// TIA Portal V18 export
FUNCTION "Re-filling Sequence" : Void   // FC14, LAD
{ S7_Optimized_Access := 'TRUE' }
VERSION : 0.1
// stored: AutoNumber true, IsIECCheckEnabled false, SetENOAutomatically false, UDAEnableTagReadback false
   VAR_TEMP   // added for the SCL form of the ladder/FBD networks
      _w1 : Bool;
      _w2 : Bool;
      _w3 : Bool;
   END_VAR
BEGIN

REGION Network 1
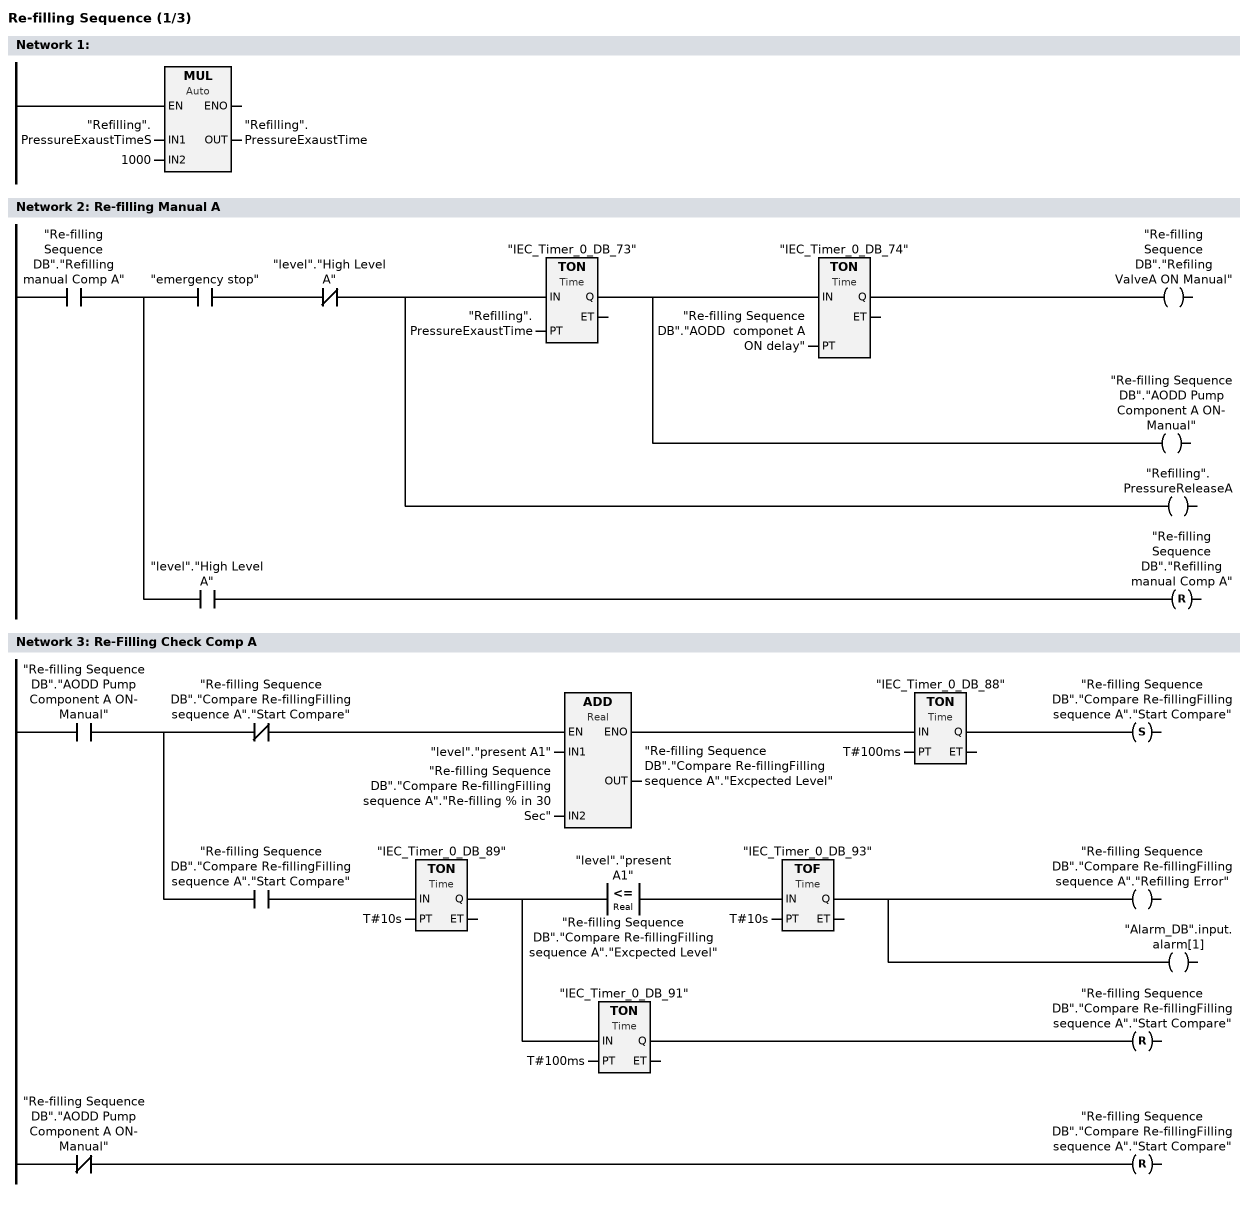
   RUNG wire#powerrail
      Mul(in1 := "Refilling".PressureExaustTimeS, in2 := 1000, out => "Refilling".PressureExaustTime)
   END_RUNG
   // the same network as SCL:
   "Refilling".PressureExaustTime := "Refilling".PressureExaustTimeS * 1000;
END_REGION

REGION Network 2: Re-filling Manual A
   RUNG wire#powerrail
      Contact( "Re-filling Sequence DB"."Refilling manual Comp A" )
      wire#w1
      Contact( "emergency stop" )
      I_Contact( "level"."High Level A" )
      wire#w2
      { S7_Templates := "time_type := Time" } "IEC_Timer_0_DB_73".TON(pt := "Refilling".PressureExaustTime, et =>)
      wire#w3
      { S7_Templates := "time_type := Time" } "IEC_Timer_0_DB_74".TON(pt := "Re-filling Sequence DB"."AODD  componet A  ON delay", et =>)
      Coil( "Re-filling Sequence DB"."Refiling ValveA ON Manual" )
   END_RUNG
   RUNG wire#w3
      Coil( "Re-filling Sequence DB"."AODD Pump Component A ON- Manual" )
   END_RUNG
   RUNG wire#w2
      Coil( "Refilling".PressureReleaseA )
   END_RUNG
   RUNG wire#w1
      Contact( "level"."High Level A" )
      R_Coil( "Re-filling Sequence DB"."Refilling manual Comp A" )
   END_RUNG
   // the same network as SCL:
   #_w1 := "Re-filling Sequence DB"."Refilling manual Comp A" AND "emergency stop" AND NOT "level"."High Level A";
   "IEC_Timer_0_DB_73".TON(IN := #_w1, PT := "Refilling".PressureExaustTime);
   "IEC_Timer_0_DB_74".TON(IN := "IEC_Timer_0_DB_73".Q,
                           PT := "Re-filling Sequence DB"."AODD  componet A  ON delay");
   "Re-filling Sequence DB"."Refiling ValveA ON Manual" := "IEC_Timer_0_DB_74".Q;
   "Re-filling Sequence DB"."AODD Pump Component A ON- Manual" := "IEC_Timer_0_DB_73".Q;
   "Refilling".PressureReleaseA := #_w1;
   IF "Re-filling Sequence DB"."Refilling manual Comp A" AND "level"."High Level A" THEN
       "Re-filling Sequence DB"."Refilling manual Comp A" := FALSE;
   END_IF;
END_REGION

REGION Network 3: Re-Filling Check Comp A
   RUNG wire#powerrail
      Contact( "Re-filling Sequence DB"."AODD Pump Component A ON- Manual" )
      wire#w1
      I_Contact( "Re-filling Sequence DB"."Compare Re-fillingFilling sequence A"."Start Compare" )
      { S7_Templates := "SrcType := Real" } Add(in1 := "level"."present A1", in2 := "Re-filling Sequence DB"."Compare Re-fillingFilling sequence A"."Re-filling % in 30 Sec", out => "Re-filling Sequence DB"."Compare Re-fillingFilling sequence A"."Excpected Level")
      { S7_Templates := "time_type := Time" } "IEC_Timer_0_DB_88".TON(pt := T#100ms, et =>)
      S_Coil( "Re-filling Sequence DB"."Compare Re-fillingFilling sequence A"."Start Compare" )
   END_RUNG
   RUNG wire#w1
      Contact( "Re-filling Sequence DB"."Compare Re-fillingFilling sequence A"."Start Compare" )
      { S7_Templates := "time_type := Time" } "IEC_Timer_0_DB_89".TON(pt := T#10s, et =>)
      wire#w2
      { S7_Templates := "SrcType := Real" } LE_Contact(in1 := "level"."present A1", in2 := "Re-filling Sequence DB"."Compare Re-fillingFilling sequence A"."Excpected Level")
      { S7_Templates := "time_type := Time" } "IEC_Timer_0_DB_93".TOF(pt := T#10s, et =>)
      wire#w3
      Coil( "Re-filling Sequence DB"."Compare Re-fillingFilling sequence A"."Refilling Error" )
   END_RUNG
   RUNG wire#w3
      Coil( "Alarm_DB".input.alarm[1] )
   END_RUNG
   RUNG wire#w2
      { S7_Templates := "time_type := Time" } "IEC_Timer_0_DB_91".TON(pt := T#100ms, et =>)
      R_Coil( "Re-filling Sequence DB"."Compare Re-fillingFilling sequence A"."Start Compare" )
   END_RUNG
   RUNG wire#powerrail
      I_Contact( "Re-filling Sequence DB"."AODD Pump Component A ON- Manual" )
      R_Coil( "Re-filling Sequence DB"."Compare Re-fillingFilling sequence A"."Start Compare" )
   END_RUNG
   // the same network as SCL:
   #_w1 := "Re-filling Sequence DB"."AODD Pump Component A ON- Manual" AND NOT "Re-filling Sequence DB"."Compare Re-fillingFilling sequence A"."Start Compare";
   IF #_w1 THEN
       "Re-filling Sequence DB"."Compare Re-fillingFilling sequence A"."Excpected Level" := "level"."present A1" + "Re-filling Sequence DB"."Compare Re-fillingFilling sequence A"."Re-filling % in 30 Sec";
   END_IF;
   "IEC_Timer_0_DB_88".TON(IN := #_w1, PT := T#100ms);
   IF "IEC_Timer_0_DB_88".Q THEN
       "Re-filling Sequence DB"."Compare Re-fillingFilling sequence A"."Start Compare" := TRUE;
   END_IF;
   "IEC_Timer_0_DB_89".TON(IN := "Re-filling Sequence DB"."AODD Pump Component A ON- Manual" AND "Re-filling Sequence DB"."Compare Re-fillingFilling sequence A"."Start Compare",
                           PT := T#10s);
   "IEC_Timer_0_DB_93".TOF(IN := "IEC_Timer_0_DB_89".Q AND ("level"."present A1" <= "Re-filling Sequence DB"."Compare Re-fillingFilling sequence A"."Excpected Level"),
                           PT := T#10s);
   "Re-filling Sequence DB"."Compare Re-fillingFilling sequence A"."Refilling Error" := "IEC_Timer_0_DB_93".Q;
   "Alarm_DB".input.alarm[1] := "IEC_Timer_0_DB_93".Q;
   "IEC_Timer_0_DB_91".TON(IN := "IEC_Timer_0_DB_89".Q, PT := T#100ms);
   IF "IEC_Timer_0_DB_91".Q THEN
       "Re-filling Sequence DB"."Compare Re-fillingFilling sequence A"."Start Compare" := FALSE;
   END_IF;
   IF NOT "Re-filling Sequence DB"."AODD Pump Component A ON- Manual" THEN
       "Re-filling Sequence DB"."Compare Re-fillingFilling sequence A"."Start Compare" := FALSE;
   END_IF;
END_REGION

REGION Network 4: Re-filling Manual B
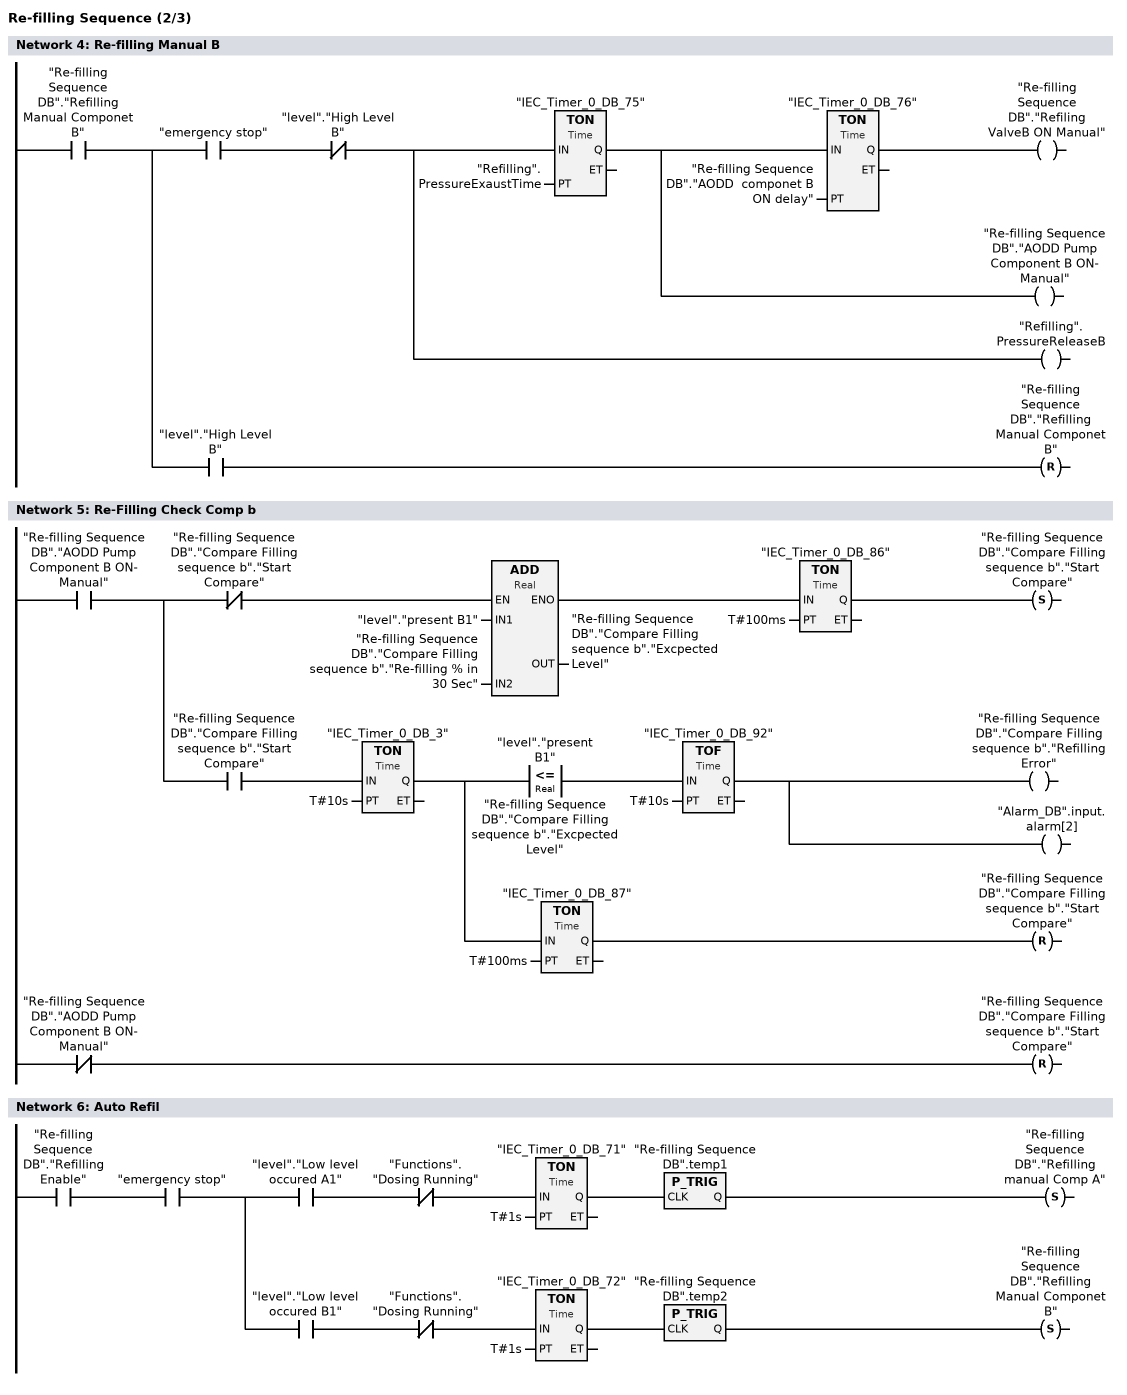
   RUNG wire#powerrail
      Contact( "Re-filling Sequence DB"."Refilling Manual Componet B" )
      wire#w1
      Contact( "emergency stop" )
      I_Contact( "level"."High Level B" )
      wire#w2
      { S7_Templates := "time_type := Time" } "IEC_Timer_0_DB_75".TON(pt := "Refilling".PressureExaustTime, et =>)
      wire#w3
      { S7_Templates := "time_type := Time" } "IEC_Timer_0_DB_76".TON(pt := "Re-filling Sequence DB"."AODD  componet B  ON delay", et =>)
      Coil( "Re-filling Sequence DB"."Refiling ValveB ON Manual" )
   END_RUNG
   RUNG wire#w3
      Coil( "Re-filling Sequence DB"."AODD Pump Component B ON- Manual" )
   END_RUNG
   RUNG wire#w2
      Coil( "Refilling".PressureReleaseB )
   END_RUNG
   RUNG wire#w1
      Contact( "level"."High Level B" )
      R_Coil( "Re-filling Sequence DB"."Refilling Manual Componet B" )
   END_RUNG
   // the same network as SCL:
   #_w1 := "Re-filling Sequence DB"."Refilling Manual Componet B" AND "emergency stop" AND NOT "level"."High Level B";
   "IEC_Timer_0_DB_75".TON(IN := #_w1, PT := "Refilling".PressureExaustTime);
   "IEC_Timer_0_DB_76".TON(IN := "IEC_Timer_0_DB_75".Q,
                           PT := "Re-filling Sequence DB"."AODD  componet B  ON delay");
   "Re-filling Sequence DB"."Refiling ValveB ON Manual" := "IEC_Timer_0_DB_76".Q;
   "Re-filling Sequence DB"."AODD Pump Component B ON- Manual" := "IEC_Timer_0_DB_75".Q;
   "Refilling".PressureReleaseB := #_w1;
   IF "Re-filling Sequence DB"."Refilling Manual Componet B" AND "level"."High Level B" THEN
       "Re-filling Sequence DB"."Refilling Manual Componet B" := FALSE;
   END_IF;
END_REGION

REGION Network 5: Re-Filling Check Comp b
   RUNG wire#powerrail
      Contact( "Re-filling Sequence DB"."AODD Pump Component B ON- Manual" )
      wire#w1
      I_Contact( "Re-filling Sequence DB"."Compare Filling sequence b"."Start Compare" )
      { S7_Templates := "SrcType := Real" } Add(in1 := "level"."present B1", in2 := "Re-filling Sequence DB"."Compare Filling sequence b"."Re-filling % in 30 Sec", out => "Re-filling Sequence DB"."Compare Filling sequence b"."Excpected Level")
      { S7_Templates := "time_type := Time" } "IEC_Timer_0_DB_86".TON(pt := T#100ms, et =>)
      S_Coil( "Re-filling Sequence DB"."Compare Filling sequence b"."Start Compare" )
   END_RUNG
   RUNG wire#w1
      Contact( "Re-filling Sequence DB"."Compare Filling sequence b"."Start Compare" )
      { S7_Templates := "time_type := Time" } "IEC_Timer_0_DB_3".TON(pt := T#10s, et =>)
      wire#w2
      { S7_Templates := "SrcType := Real" } LE_Contact(in1 := "level"."present B1", in2 := "Re-filling Sequence DB"."Compare Filling sequence b"."Excpected Level")
      { S7_Templates := "time_type := Time" } "IEC_Timer_0_DB_92".TOF(pt := T#10s, et =>)
      wire#w3
      Coil( "Re-filling Sequence DB"."Compare Filling sequence b"."Refilling Error" )
   END_RUNG
   RUNG wire#w3
      Coil( "Alarm_DB".input.alarm[2] )
   END_RUNG
   RUNG wire#w2
      { S7_Templates := "time_type := Time" } "IEC_Timer_0_DB_87".TON(pt := T#100ms, et =>)
      R_Coil( "Re-filling Sequence DB"."Compare Filling sequence b"."Start Compare" )
   END_RUNG
   RUNG wire#powerrail
      I_Contact( "Re-filling Sequence DB"."AODD Pump Component B ON- Manual" )
      R_Coil( "Re-filling Sequence DB"."Compare Filling sequence b"."Start Compare" )
   END_RUNG
   // the same network as SCL:
   #_w1 := "Re-filling Sequence DB"."AODD Pump Component B ON- Manual" AND NOT "Re-filling Sequence DB"."Compare Filling sequence b"."Start Compare";
   IF #_w1 THEN
       "Re-filling Sequence DB"."Compare Filling sequence b"."Excpected Level" := "level"."present B1" + "Re-filling Sequence DB"."Compare Filling sequence b"."Re-filling % in 30 Sec";
   END_IF;
   "IEC_Timer_0_DB_86".TON(IN := #_w1, PT := T#100ms);
   IF "IEC_Timer_0_DB_86".Q THEN
       "Re-filling Sequence DB"."Compare Filling sequence b"."Start Compare" := TRUE;
   END_IF;
   "IEC_Timer_0_DB_3".TON(IN := "Re-filling Sequence DB"."AODD Pump Component B ON- Manual" AND "Re-filling Sequence DB"."Compare Filling sequence b"."Start Compare",
                          PT := T#10s);
   "IEC_Timer_0_DB_92".TOF(IN := "IEC_Timer_0_DB_3".Q AND ("level"."present B1" <= "Re-filling Sequence DB"."Compare Filling sequence b"."Excpected Level"),
                           PT := T#10s);
   "Re-filling Sequence DB"."Compare Filling sequence b"."Refilling Error" := "IEC_Timer_0_DB_92".Q;
   "Alarm_DB".input.alarm[2] := "IEC_Timer_0_DB_92".Q;
   "IEC_Timer_0_DB_87".TON(IN := "IEC_Timer_0_DB_3".Q, PT := T#100ms);
   IF "IEC_Timer_0_DB_87".Q THEN
       "Re-filling Sequence DB"."Compare Filling sequence b"."Start Compare" := FALSE;
   END_IF;
   IF NOT "Re-filling Sequence DB"."AODD Pump Component B ON- Manual" THEN
       "Re-filling Sequence DB"."Compare Filling sequence b"."Start Compare" := FALSE;
   END_IF;
END_REGION

REGION Network 6: Auto Refil
   RUNG wire#powerrail
      Contact( "Re-filling Sequence DB"."Refilling Enable" )
      Contact( "emergency stop" )
      wire#w1
      Contact( "level"."Low level occured A1" )
      I_Contact( "Functions"."Dosing Running" )
      { S7_Templates := "time_type := Time" } "IEC_Timer_0_DB_71".TON(pt := T#1s, et =>)
      P_Trig( "Re-filling Sequence DB".temp1 )
      S_Coil( "Re-filling Sequence DB"."Refilling manual Comp A" )
   END_RUNG
   RUNG wire#w1
      Contact( "level"."Low level occured B1" )
      I_Contact( "Functions"."Dosing Running" )
      { S7_Templates := "time_type := Time" } "IEC_Timer_0_DB_72".TON(pt := T#1s, et =>)
      P_Trig( "Re-filling Sequence DB".temp2 )
      S_Coil( "Re-filling Sequence DB"."Refilling Manual Componet B" )
   END_RUNG
   // the same network as SCL:
   #_w1 := "Re-filling Sequence DB"."Refilling Enable" AND "emergency stop";
   "IEC_Timer_0_DB_71".TON(IN := #_w1 AND "level"."Low level occured A1" AND NOT "Functions"."Dosing Running",
                           PT := T#1s);
   #_w2 := "IEC_Timer_0_DB_71".Q AND NOT "Re-filling Sequence DB".temp1;   // rising edge
   "Re-filling Sequence DB".temp1 := "IEC_Timer_0_DB_71".Q;
   IF #_w2 THEN "Re-filling Sequence DB"."Refilling manual Comp A" := TRUE; END_IF;
   "IEC_Timer_0_DB_72".TON(IN := #_w1 AND "level"."Low level occured B1" AND NOT "Functions"."Dosing Running",
                           PT := T#1s);
   #_w3 := "IEC_Timer_0_DB_72".Q AND NOT "Re-filling Sequence DB".temp2;   // rising edge
   "Re-filling Sequence DB".temp2 := "IEC_Timer_0_DB_72".Q;
   IF #_w3 THEN "Re-filling Sequence DB"."Refilling Manual Componet B" := TRUE; END_IF;
END_REGION

REGION Network 7: Auto reffil reset
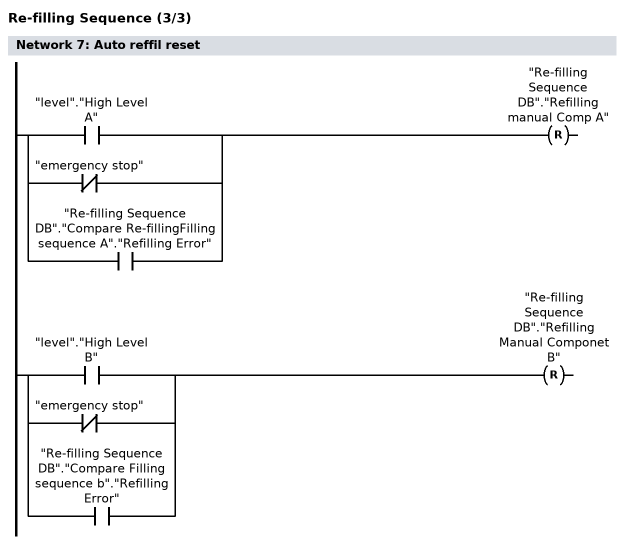
   RUNG wire#powerrail
      Contact( "level"."High Level A" )
      wire#w1
      R_Coil( "Re-filling Sequence DB"."Refilling manual Comp A" )
   END_RUNG
   RUNG wire#powerrail
      I_Contact( "emergency stop" )
   END_RUNG wire#w1
   RUNG wire#powerrail
      Contact( "Re-filling Sequence DB"."Compare Re-fillingFilling sequence A"."Refilling Error" )
   END_RUNG wire#w1
   RUNG wire#powerrail
      Contact( "level"."High Level B" )
      wire#w2
      R_Coil( "Re-filling Sequence DB"."Refilling Manual Componet B" )
   END_RUNG
   RUNG wire#powerrail
      I_Contact( "emergency stop" )
   END_RUNG wire#w2
   RUNG wire#powerrail
      Contact( "Re-filling Sequence DB"."Compare Filling sequence b"."Refilling Error" )
   END_RUNG wire#w2
   // the same network as SCL:
   IF "level"."High Level A" OR NOT "emergency stop" OR "Re-filling Sequence DB"."Compare Re-fillingFilling sequence A"."Refilling Error" THEN
       "Re-filling Sequence DB"."Refilling manual Comp A" := FALSE;
   END_IF;
   IF "level"."High Level B" OR NOT "emergency stop" OR "Re-filling Sequence DB"."Compare Filling sequence b"."Refilling Error" THEN
       "Re-filling Sequence DB"."Refilling Manual Componet B" := FALSE;
   END_IF;
END_REGION
END_FUNCTION
